(* Logix 5000 project; controller cal1615 1756-L62 rev 20.19; software revision 20.05; part 58 of 82 *)
(* tags used below, declared in another part *)
   FAULT : BOOL;   // Fault AFI
   p01_recipe_active : recipe;   // Active Recipe
   p01r02 : routine;   // System Misc Control
   p01r09_pb_global_reset : BOOL;   // System Modes PB: Global Fault Reset
   p24_di_edge_guide_auto : BOOL;   // Edge Control Inputs SS: Edge Guide Manual/Auto Auto
   p24_di_edge_guide_center : BOOL;   // Edge Control Inputs PB: Edge Guide Center
   p24_di_edge_guide_left : BOOL;   // Edge Control Inputs PB: Edge Guide Left
   p24_di_edge_guide_right : BOOL;   // Edge Control Inputs PB: Edge Guide Right
   p24_do_edge_guide_input_1 : BOOL;   // Edge Guide Digital Output Input 1
   p24_do_edge_guide_input_2 : BOOL;   // Edge Guide Digital Output Input 2
   p24_do_edge_guide_input_3 : BOOL;   // Edge Guide Digital Output Input 3
   p24_do_edge_guide_input_4 : BOOL;   // Edge Guide Digital Output Input 4
   p24_do_edge_guide_input_5 : BOOL;   // Edge Guide Digital Output Input 5
   p24r01 : routine;
   p24r10 : routine;   // Edge Control Edge Guide
   p24r10_edge_guide_auto_request : BOOL;   // Edge Control Edge Guide Auto Request
   p24r10_edge_guide_center_request : BOOL;   // Edge Control Edge Guide Center Request
   p24r10_edge_guide_jog_left_request : BOOL;   // Edge Control Edge Guide Jog Left Request
   p24r10_edge_guide_jog_right_request : BOOL;   // Edge Control Edge Guide Jog Right Request
   p24r10_timer_fault : TIMER[4];   // Edge Control Edge Guide Fault Delay
   p24r10_timer_warning : TIMER[4];   // Edge Control Edge Guide Warning Delay
   p25_ai_amps : DINT;   // Tension Stand 2 Analog Input TS 2 Motor Current
   p25_ai_hz : DINT;   // Tension Stand 2 Analog Input TS 2 Motor Hertz
   p25_ai_speed : REAL;   // Tension Stand 2 Inputs Sufrace Speed [fpm]
   p25_ai_torque : REAL;
   p25_ai_ts2_lc : REAL;   // System Metering Roll VFD Minimum Start Tension
   p25_di_brake : BOOL;   // Tension Stand 2 Digital Input TS2 & Slitter Brake Temperature OK
   p25_di_jog : BOOL;   // Tension Stand 2 Digital Input SS: Jog
   p25_di_jog_fwd : BOOL;   // Tension Stand 2 Digital Input PB: Jog Forward
   p25_di_jog_rev : BOOL;   // Tension Stand 2 Digital Input PB: Jog Reverse
   p25_di_run : BOOL;   // Tension Stand 2 Digital Input SS: Run
   p25_di_therm : BOOL;   // Tension Stand 2 Digital Input Motor Temperature OK
   p25_dint_to_hmi : DINT[16];   // Tension Stand 2 Dint to HMI
   p25_param_payout_speed_factor : REAL;   // Tension Stand 2 Accumulator Payout Winder Overspeed Factor 0.20 = 1.20 x Line Speed
   p25_status_word : INT;
   p25_ts2_gear_ratio : REAL;
   p25_ts2_roll_diameter_ft : REAL;
   p25r01 : routine;
   p25r02 : routine;
   p25r02_fault_exists : BOOL;
   p25r02_tension_dev_max : REAL;
   p25r02_tension_dev_min : REAL;
   p25r02_timer_fault : TIMER[4];   // Tension Stand 2 Misc Control Fault Dwell Timer
   p25r02_timer_warning : TIMER[4];   // Tension Stand 2 Misc Control Warning Dwell Timer
   p25r02_unack_fault : BOOL;   // Upper Poly Letoff Misc Control Unacknowledged Fault Exists
   p25r02_unack_warning : BOOL;   // Upper Poly Letoff Misc Control Unacknowledged Warning Exists
   p25r02_warning_exists : BOOL;
   p25r03 : routine;
   p25r03_ave_tq : REAL;
   p25r03_hz : SYS_SCP;   // Tension Stand 2 Analog Inputs SCP Hz
   p25r03_lc_input_max : REAL;
   p25r03_lc_input_min : REAL;
   p25r03_lc_output_max : REAL;
   p25r03_lc_output_min : REAL;
   p25r03_lc_scp : SYS_SCP;   // Tension Stand 2 Analog Input Load Cell Scaling
   p25r03_sample_timer : TIMER;
   p25r03_scaled_vfd_in : REAL;
   p25r03_timer_fault : TIMER[4];   // Tension Stand 2 Inputs Fault Dwell Timer
   p25r03_timer_warning : TIMER[4];   // Tension Stand 2 Inputs Warning Dwell Timer
   p25r03_tq_ave_ctrl : CONTROL;
   p25r03_tq_buffer : REAL[20];
   p25r03_tq_fifo : CONTROL;
   p25R03_ts2_vfd_rpm_to_speed : SYS_RPM_TO_SPEED;   // Tension Stand 2 Analog Input VFD RPM to Roll Surface Speed
   p25r03_unload : DINT;
   p25r03_vfd_in_scaling : SYS_SCP;
   p25r03_vfd_input_max : REAL;
   p25r03_vfd_input_min : REAL;
   p25r03_vfd_output_max : REAL;
   p25r03_vfd_output_min : REAL;
   p25r04 : routine;
   p25r05 : routine;
   p25r06 : routine;
   p25r07 : routine;
   p25r08 : routine;
   p25r09 : routine;   // Upper Poly Letoff Modes
   p25r10 : routine;
   p25r11 : routine;   // Tension Stand 2 VFD
(* P24_Edge_Control, continued *)

ROUTINE R10_Edge_Guide   (* ladder *)
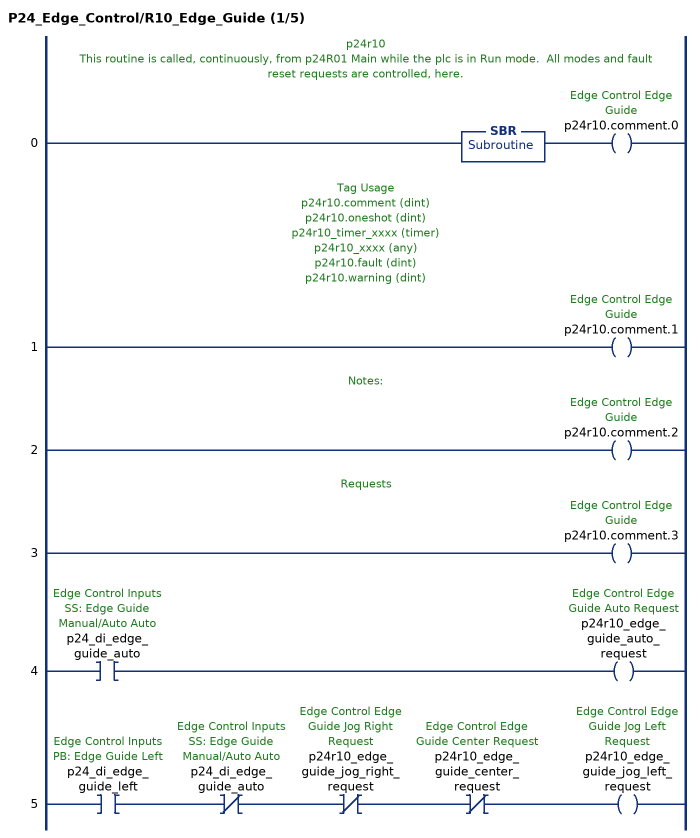
   // p24r10
   // This routine is called, continuously, from p24R01 Main while the plc is in Run mode.  All modes and fault reset requests are controlled, here.
   0: SBR()OTE(p24r10.comment.0);
   // Tag Usage
   // p24r10.comment (dint)
   // p24r10.oneshot (dint)
   // p24r10_timer_xxxx (timer)
   // p24r10_xxxx (any)
   // p24r10.fault (dint)
   // p24r10.warning (dint)
   1: OTE(p24r10.comment.1);
   // Notes:
   2: OTE(p24r10.comment.2);
   // Requests
   3: OTE(p24r10.comment.3);
   4: XIC(p24_di_edge_guide_auto)OTE(p24r10_edge_guide_auto_request);
   5: XIC(p24_di_edge_guide_left)XIO(p24_di_edge_guide_auto)XIO(p24r10_edge_guide_jog_right_request)XIO(p24r10_edge_guide_center_request)OTE(p24r10_edge_guide_jog_left_request);
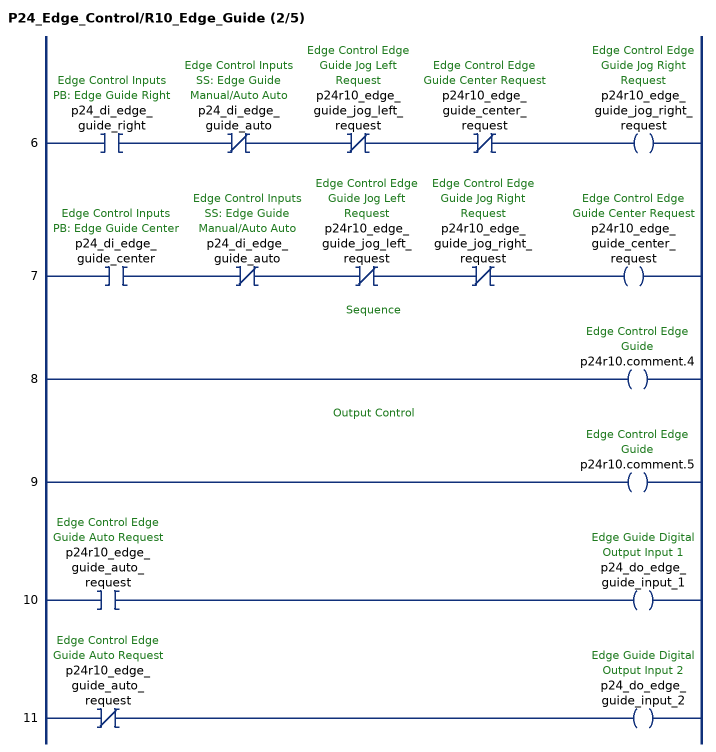
   6: XIC(p24_di_edge_guide_right)XIO(p24_di_edge_guide_auto)XIO(p24r10_edge_guide_jog_left_request)XIO(p24r10_edge_guide_center_request)OTE(p24r10_edge_guide_jog_right_request);
   7: XIC(p24_di_edge_guide_center)XIO(p24_di_edge_guide_auto)XIO(p24r10_edge_guide_jog_left_request)XIO(p24r10_edge_guide_jog_right_request)OTE(p24r10_edge_guide_center_request);
   // Sequence
   8: OTE(p24r10.comment.4);
   // Output Control
   9: OTE(p24r10.comment.5);
   10: XIC(p24r10_edge_guide_auto_request)OTE(p24_do_edge_guide_input_1);
   11: XIO(p24r10_edge_guide_auto_request)OTE(p24_do_edge_guide_input_2);
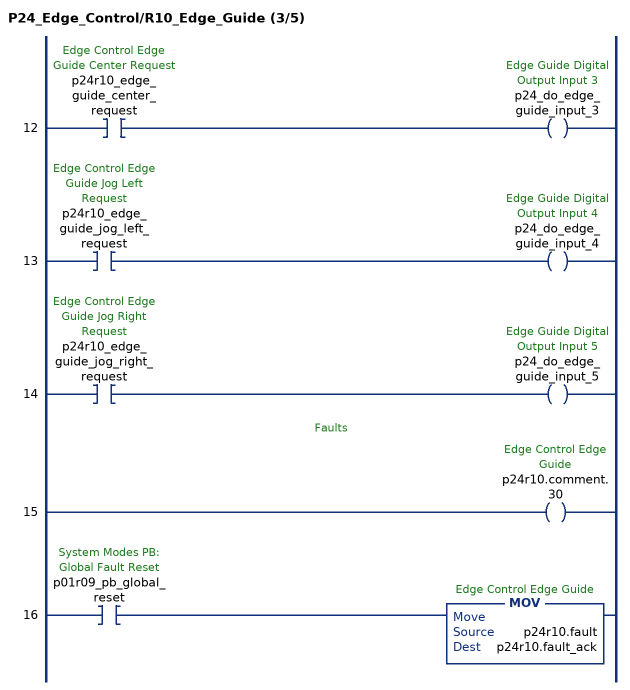
   12: XIC(p24r10_edge_guide_center_request)OTE(p24_do_edge_guide_input_3);
   13: XIC(p24r10_edge_guide_jog_left_request)OTE(p24_do_edge_guide_input_4);
   14: XIC(p24r10_edge_guide_jog_right_request)OTE(p24_do_edge_guide_input_5);
   // Faults
   15: OTE(p24r10.comment.30);
   16: XIC(p01r09_pb_global_reset)MOV(p24r10.fault,p24r10.fault_ack);
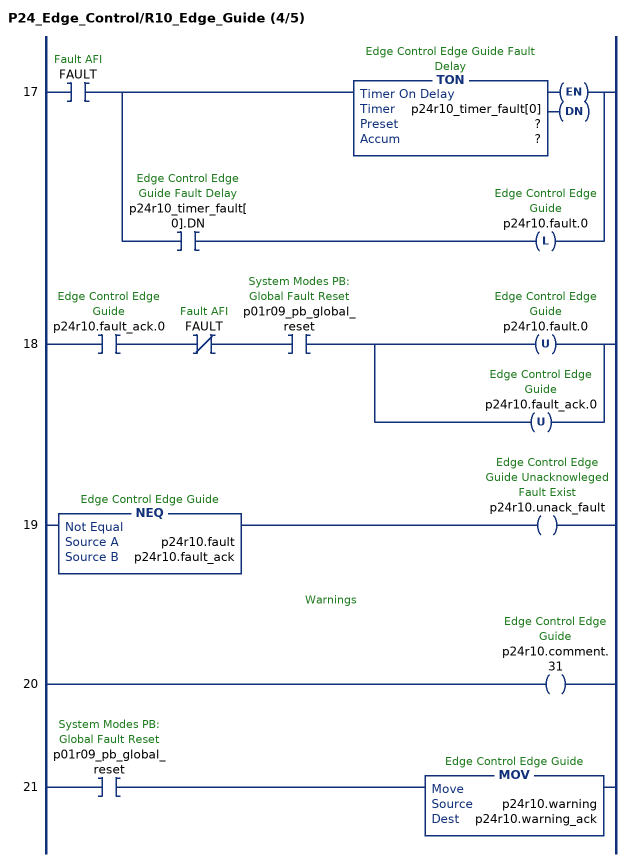
   17: XIC(FAULT)[TON(p24r10_timer_fault[0],?,?) ,XIC(p24r10_timer_fault[0].DN) OTL(p24r10.fault.0) ];
   18: XIC(p24r10.fault_ack.0)XIO(FAULT)XIC(p01r09_pb_global_reset)[OTU(p24r10.fault.0) ,OTU(p24r10.fault_ack.0) ];
   19: NEQ(p24r10.fault,p24r10.fault_ack)OTE(p24r10.unack_fault);
   // Warnings
   20: OTE(p24r10.comment.31);
   21: XIC(p01r09_pb_global_reset)MOV(p24r10.warning,p24r10.warning_ack);
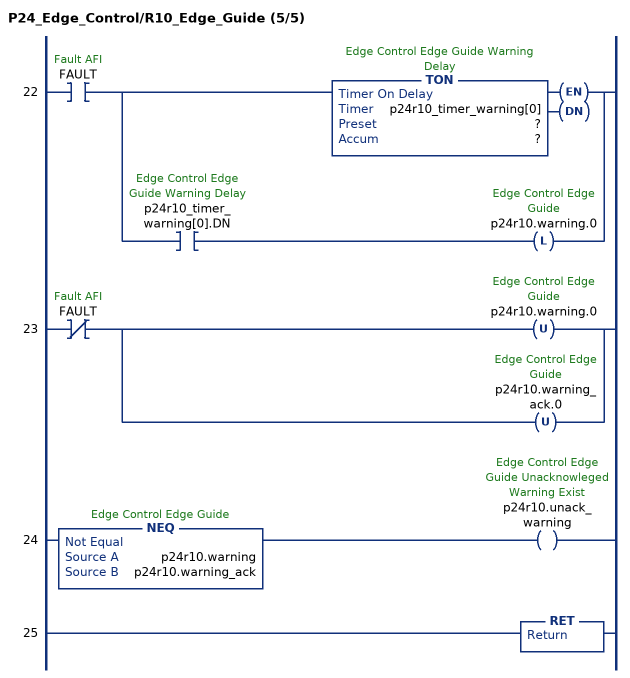
   22: XIC(FAULT)[TON(p24r10_timer_warning[0],?,?) ,XIC(p24r10_timer_warning[0].DN) OTL(p24r10.warning.0) ];
   23: XIO(FAULT)[OTU(p24r10.warning.0) ,OTU(p24r10.warning_ack.0) ];
   24: NEQ(p24r10.warning,p24r10.warning_ack)OTE(p24r10.unack_warning);
   25: RET();
END_ROUTINE
END_PROGRAM

PROGRAM P25_Tension_Stand_2   (* main routine R01_Main *)
VAR
   param_payout_speed : Setpoint := (SP := 0.2, Hi := 1.0);
   sys_limit_clamp : sys_Limit_Clamp := (max := 1.0);
END_VAR

ROUTINE R01_Main   (* ladder *)
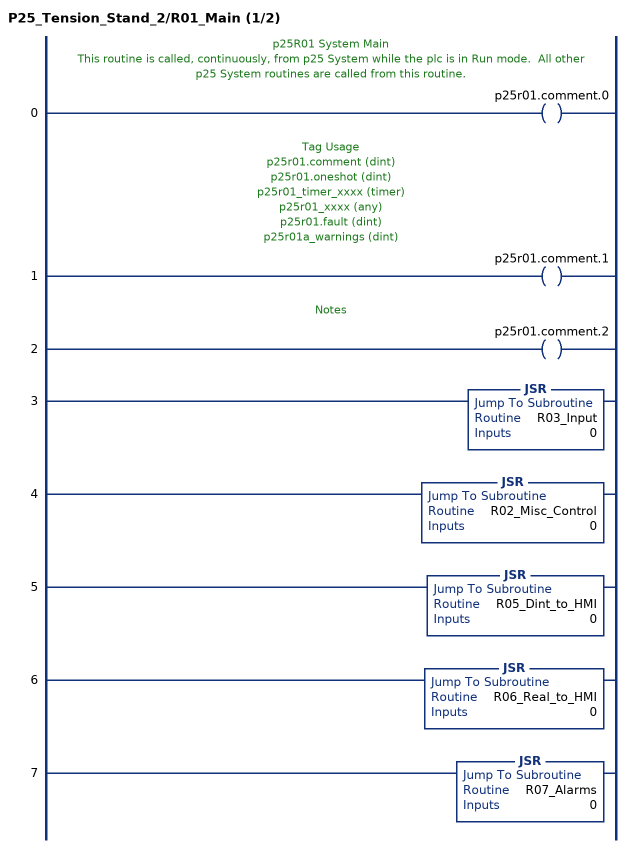
   // p25R01 System Main
   // This routine is called, continuously, from p25 System while the plc is in Run mode.  All other p25 System routines are called from this routine.
   0: OTE(p25r01.comment.0);
   // Tag Usage
   // p25r01.comment (dint)
   // p25r01.oneshot (dint)
   // p25r01_timer_xxxx (timer)
   // p25r01_xxxx (any)
   // p25r01.fault (dint)
   // p25r01a_warnings (dint)
   1: OTE(p25r01.comment.1);
   // Notes
   2: OTE(p25r01.comment.2);
   3: JSR(R03_Input,0);
   4: JSR(R02_Misc_Control,0);
   5: JSR(R05_Dint_to_HMI,0);
   6: JSR(R06_Real_to_HMI,0);
   7: JSR(R07_Alarms,0);
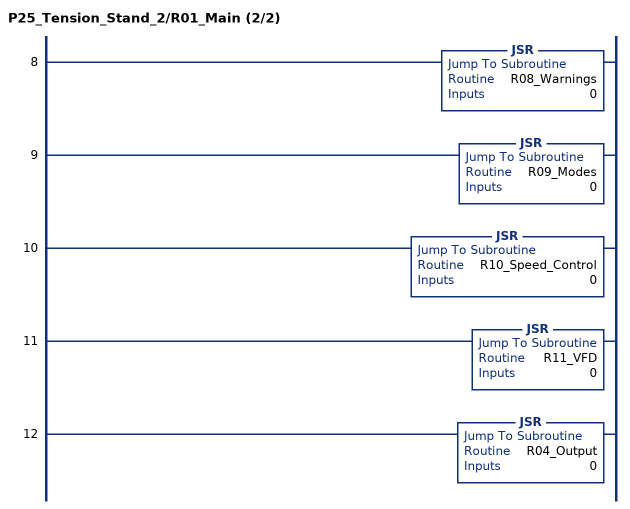
   8: JSR(R08_Warnings,0);
   9: JSR(R09_Modes,0);
   10: JSR(R10_Speed_Control,0);
   11: JSR(R11_VFD,0);
   12: JSR(R04_Output,0);
END_ROUTINE

ROUTINE R02_Misc_Control   (* ladder *)
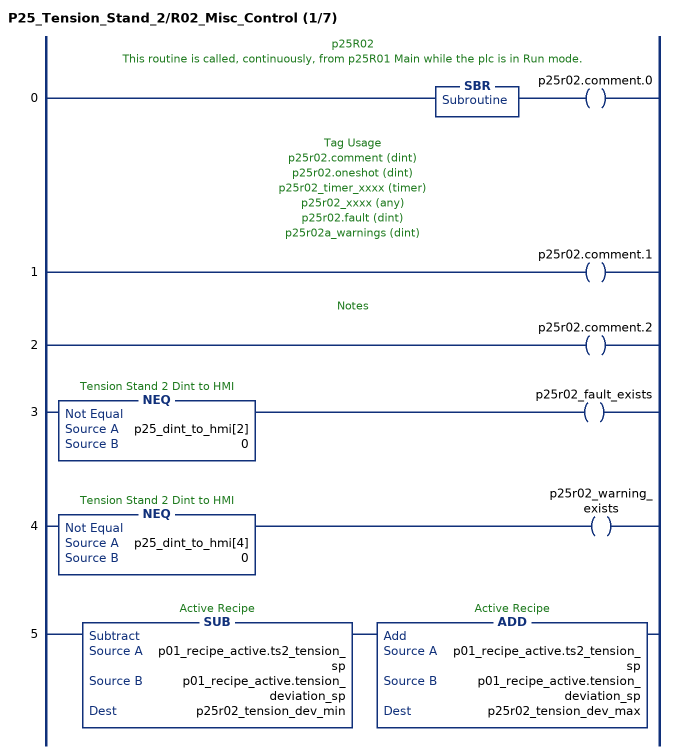
   // p25R02
   // This routine is called, continuously, from p25R01 Main while the plc is in Run mode.
   0: SBR()OTE(p25r02.comment.0);
   // Tag Usage
   // p25r02.comment (dint)
   // p25r02.oneshot (dint)
   // p25r02_timer_xxxx (timer)
   // p25r02_xxxx (any)
   // p25r02.fault (dint)
   // p25r02a_warnings (dint)
   1: OTE(p25r02.comment.1);
   // Notes
   2: OTE(p25r02.comment.2);
   3: NEQ(p25_dint_to_hmi[2],0)OTE(p25r02_fault_exists);
   4: NEQ(p25_dint_to_hmi[4],0)OTE(p25r02_warning_exists);
   5: SUB(p01_recipe_active.ts2_tension_sp,p01_recipe_active.tension_deviation_sp,p25r02_tension_dev_min)ADD(p01_recipe_active.ts2_tension_sp,p01_recipe_active.tension_deviation_sp,p25r02_tension_dev_max);
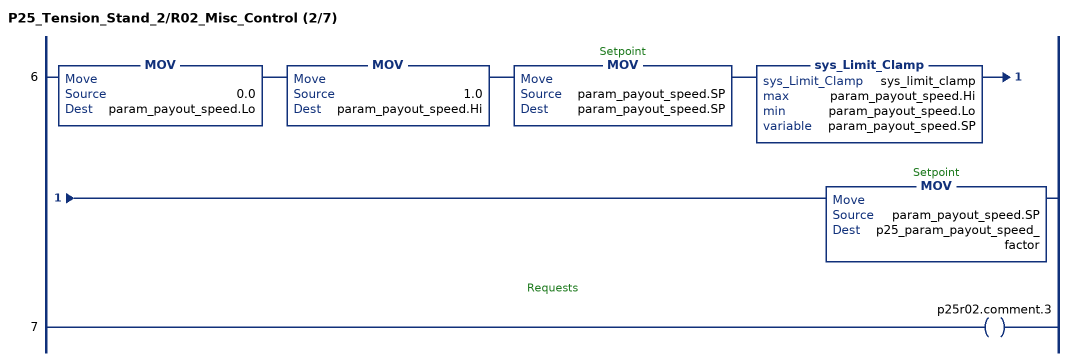
   6: MOV(0.0,param_payout_speed.Lo)MOV(1.0,param_payout_speed.Hi)MOV(param_payout_speed.SP,param_payout_speed.SP)sys_Limit_Clamp(sys_limit_clamp,param_payout_speed.Hi,param_payout_speed.Lo,param_payout_speed.SP)MOV(param_payout_speed.SP,p25_param_payout_speed_factor);
   // Requests
   7: OTE(p25r02.comment.3);
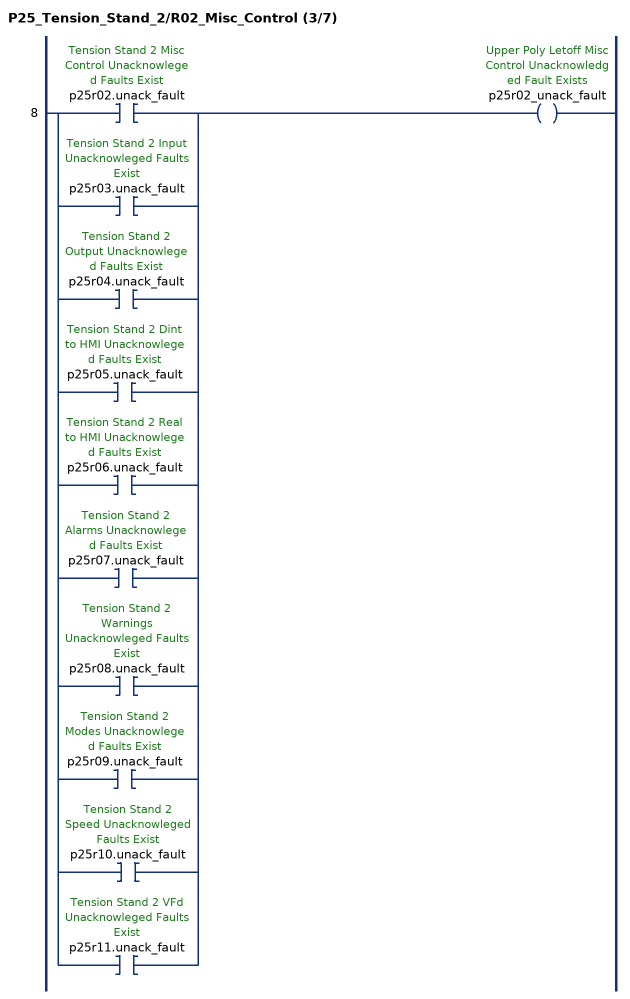
   8: [XIC(p25r02.unack_fault) ,XIC(p25r03.unack_fault) ,XIC(p25r04.unack_fault) ,XIC(p25r05.unack_fault) ,XIC(p25r06.unack_fault) ,XIC(p25r07.unack_fault) ,XIC(p25r08.unack_fault) ,XIC(p25r09.unack_fault) ,XIC(p25r10.unack_fault) ,XIC(p25r11.unack_fault) ]OTE(p25r02_unack_fault);
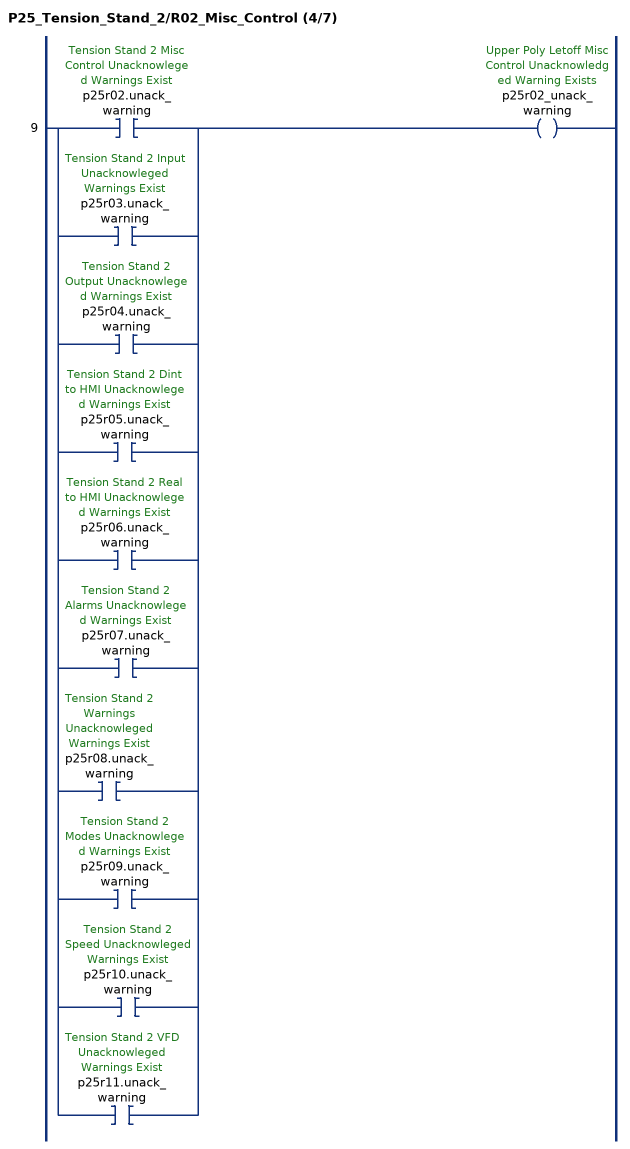
   9: [XIC(p25r02.unack_warning) ,XIC(p25r03.unack_warning) ,XIC(p25r04.unack_warning) ,XIC(p25r05.unack_warning) ,XIC(p25r06.unack_warning) ,XIC(p25r07.unack_warning) ,XIC(p25r08.unack_warning) ,XIC(p25r09.unack_warning) ,XIC(p25r10.unack_warning) ,XIC(p25r11.unack_warning) ]OTE(p25r02_unack_warning);
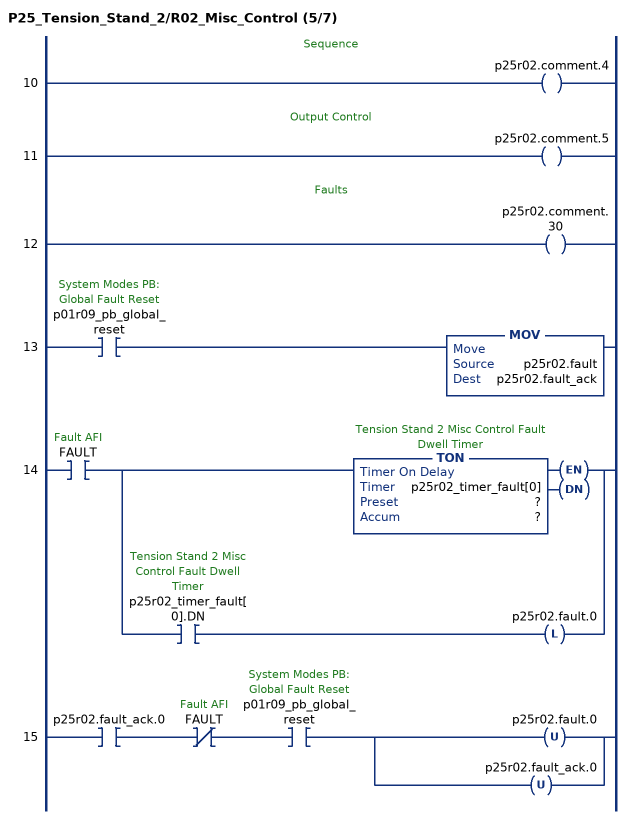
   // Sequence
   10: OTE(p25r02.comment.4);
   // Output Control
   11: OTE(p25r02.comment.5);
   // Faults
   12: OTE(p25r02.comment.30);
   13: XIC(p01r09_pb_global_reset)MOV(p25r02.fault,p25r02.fault_ack);
   14: XIC(FAULT)[TON(p25r02_timer_fault[0],?,?) ,XIC(p25r02_timer_fault[0].DN) OTL(p25r02.fault.0) ];
   15: XIC(p25r02.fault_ack.0)XIO(FAULT)XIC(p01r09_pb_global_reset)[OTU(p25r02.fault.0) ,OTU(p25r02.fault_ack.0) ];
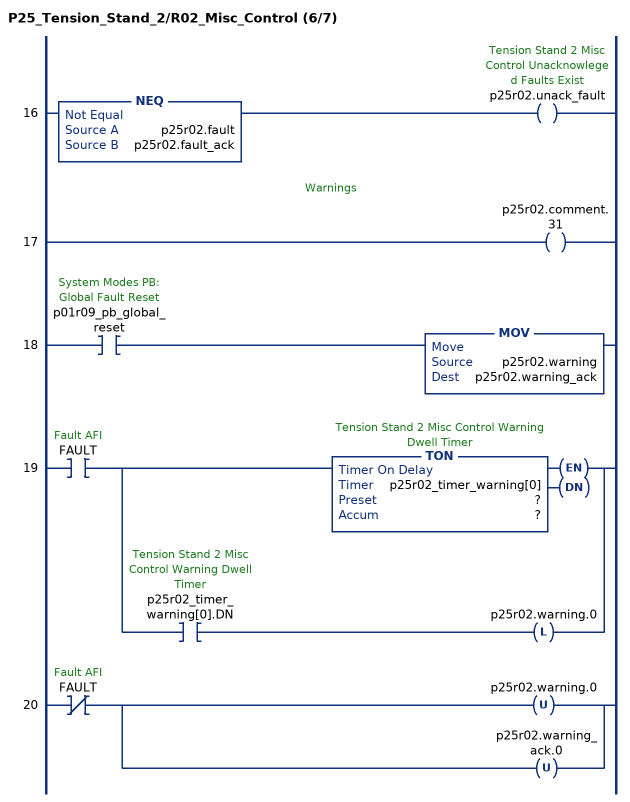
   16: NEQ(p25r02.fault,p25r02.fault_ack)OTE(p25r02.unack_fault);
   // Warnings
   17: OTE(p25r02.comment.31);
   18: XIC(p01r09_pb_global_reset)MOV(p25r02.warning,p25r02.warning_ack);
   19: XIC(FAULT)[TON(p25r02_timer_warning[0],?,?) ,XIC(p25r02_timer_warning[0].DN) OTL(p25r02.warning.0) ];
   20: XIO(FAULT)[OTU(p25r02.warning.0) ,OTU(p25r02.warning_ack.0) ];
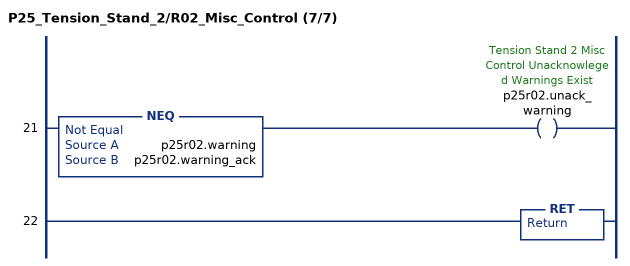
   21: NEQ(p25r02.warning,p25r02.warning_ack)OTE(p25r02.unack_warning);
   22: RET();
END_ROUTINE

ROUTINE R03_Input   (* ladder *)
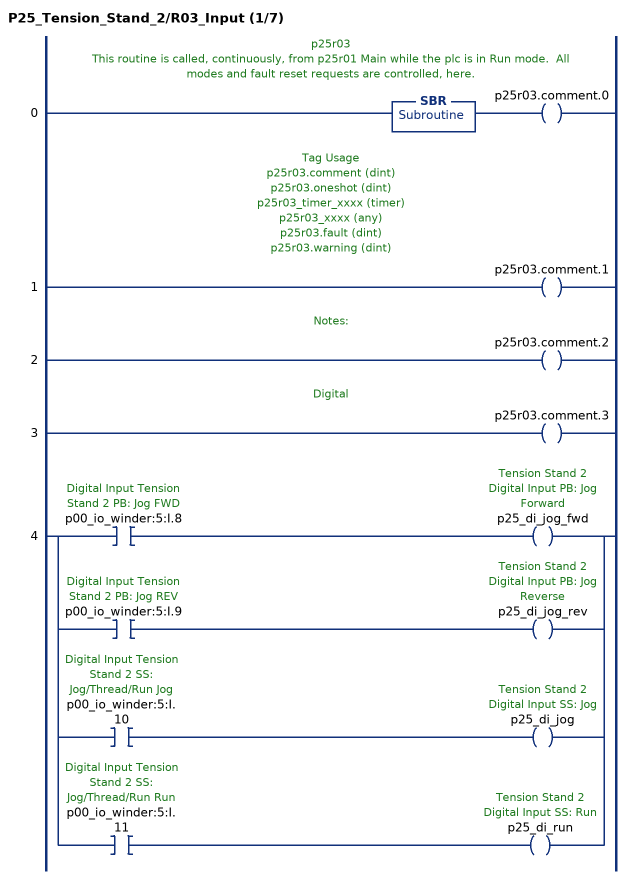
   // p25r03
   // This routine is called, continuously, from p25r01 Main while the plc is in Run mode.  All modes and fault reset requests are controlled, here.
   0: SBR()OTE(p25r03.comment.0);
   // Tag Usage
   // p25r03.comment (dint)
   // p25r03.oneshot (dint)
   // p25r03_timer_xxxx (timer)
   // p25r03_xxxx (any)
   // p25r03.fault (dint)
   // p25r03.warning (dint)
   1: OTE(p25r03.comment.1);
   // Notes:
   2: OTE(p25r03.comment.2);
   // Digital
   3: OTE(p25r03.comment.3);
   4: [XIC(p00_io_winder:5:I.8) OTE(p25_di_jog_fwd) ,XIC(p00_io_winder:5:I.9) OTE(p25_di_jog_rev) ,XIC(p00_io_winder:5:I.10) OTE(p25_di_jog) ,XIC(p00_io_winder:5:I.11) OTE(p25_di_run) ];
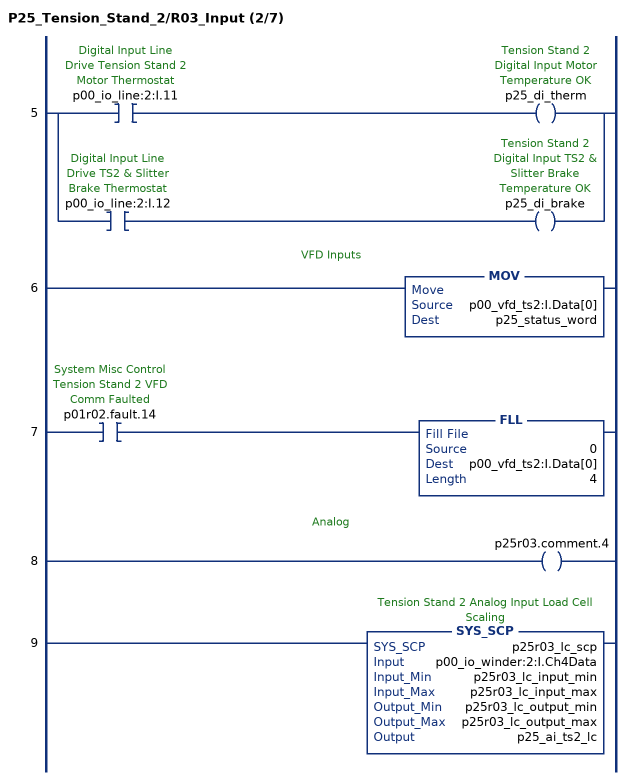
   5: [XIC(p00_io_line:2:I.11) OTE(p25_di_therm) ,XIC(p00_io_line:2:I.12) OTE(p25_di_brake) ];
   // VFD Inputs
   6: MOV(p00_vfd_ts2:I.Data[0],p25_status_word);
   7: XIC(p01r02.fault.14)FLL(0,p00_vfd_ts2:I.Data[0],4);
   // Analog
   8: OTE(p25r03.comment.4);
   9: SYS_SCP(p25r03_lc_scp,p00_io_winder:2:I.Ch4Data,p25r03_lc_input_min,p25r03_lc_input_max,p25r03_lc_output_min,p25r03_lc_output_max,p25_ai_ts2_lc);
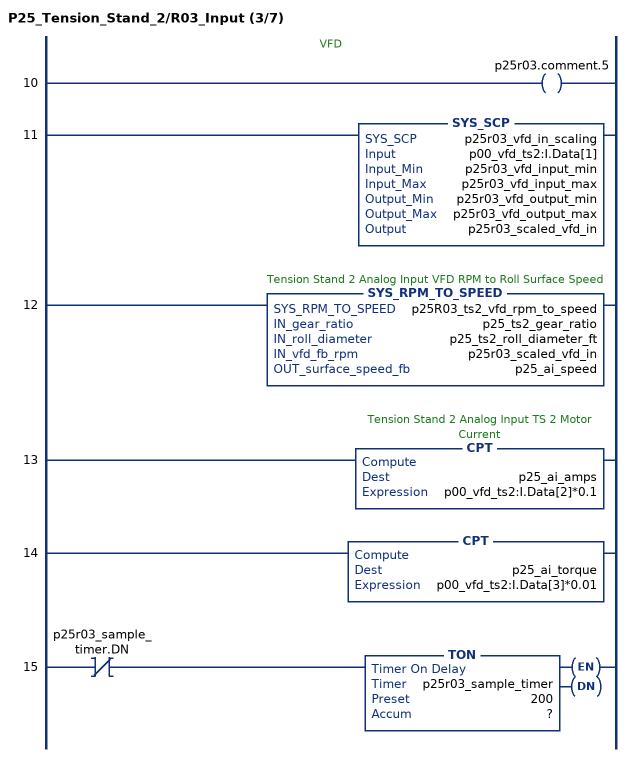
   // VFD
   10: OTE(p25r03.comment.5);
   11: SYS_SCP(p25r03_vfd_in_scaling,p00_vfd_ts2:I.Data[1],p25r03_vfd_input_min,p25r03_vfd_input_max,p25r03_vfd_output_min,p25r03_vfd_output_max,p25r03_scaled_vfd_in);
   12: SYS_RPM_TO_SPEED(p25R03_ts2_vfd_rpm_to_speed,p25_ts2_gear_ratio,p25_ts2_roll_diameter_ft,p25r03_scaled_vfd_in,p25_ai_speed);
   13: CPT(p25_ai_amps,p00_vfd_ts2:I.Data[2]*0.1);
   14: CPT(p25_ai_torque,p00_vfd_ts2:I.Data[3]*0.01);
   15: XIO(p25r03_sample_timer.DN)TON(p25r03_sample_timer,?,?);
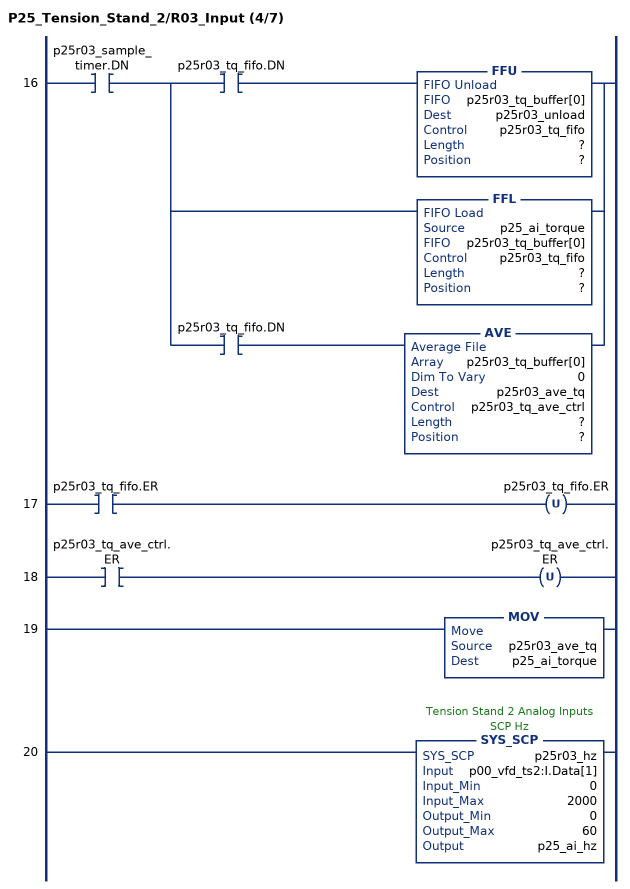
   16: XIC(p25r03_sample_timer.DN)[XIC(p25r03_tq_fifo.DN) FFU(p25r03_tq_buffer[0],p25r03_unload,p25r03_tq_fifo,?,?) ,FFL(p25_ai_torque,p25r03_tq_buffer[0],p25r03_tq_fifo,?,?) ,XIC(p25r03_tq_fifo.DN) AVE(p25r03_tq_buffer[0],0,p25r03_ave_tq,p25r03_tq_ave_ctrl,?,?) ];
   17: XIC(p25r03_tq_fifo.ER)OTU(p25r03_tq_fifo.ER);
   18: XIC(p25r03_tq_ave_ctrl.ER)OTU(p25r03_tq_ave_ctrl.ER);
   19: MOV(p25r03_ave_tq,p25_ai_torque);
   20: SYS_SCP(p25r03_hz,p00_vfd_ts2:I.Data[1],0,2000,0,60,p25_ai_hz);
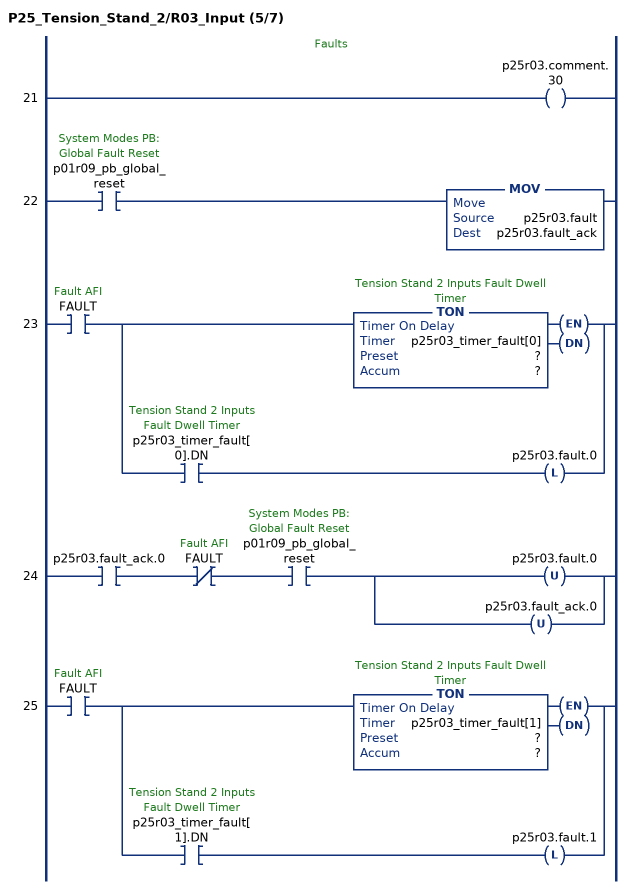
   // Faults
   21: OTE(p25r03.comment.30);
   22: XIC(p01r09_pb_global_reset)MOV(p25r03.fault,p25r03.fault_ack);
   23: XIC(FAULT)[TON(p25r03_timer_fault[0],?,?) ,XIC(p25r03_timer_fault[0].DN) OTL(p25r03.fault.0) ];
   24: XIC(p25r03.fault_ack.0)XIO(FAULT)XIC(p01r09_pb_global_reset)[OTU(p25r03.fault.0) ,OTU(p25r03.fault_ack.0) ];
   25: XIC(FAULT)[TON(p25r03_timer_fault[1],?,?) ,XIC(p25r03_timer_fault[1].DN) OTL(p25r03.fault.1) ];
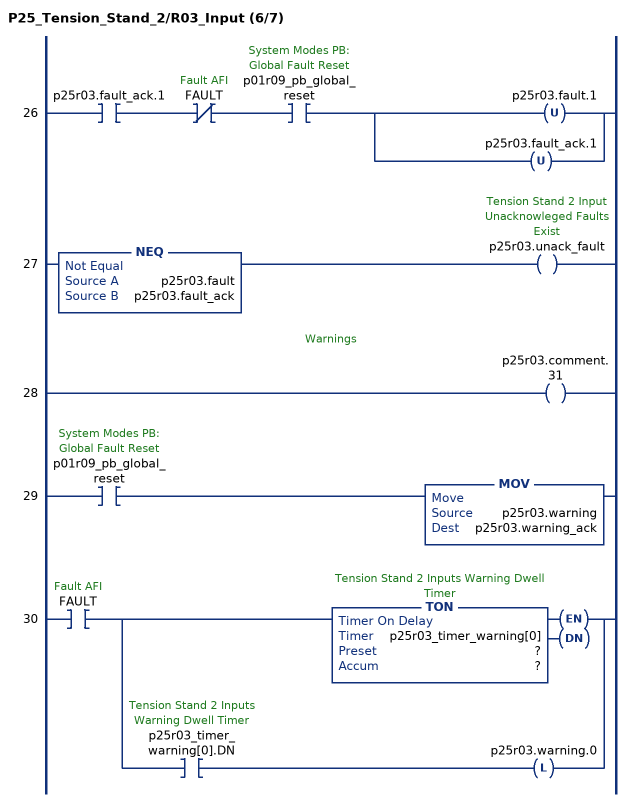
   26: XIC(p25r03.fault_ack.1)XIO(FAULT)XIC(p01r09_pb_global_reset)[OTU(p25r03.fault.1) ,OTU(p25r03.fault_ack.1) ];
   27: NEQ(p25r03.fault,p25r03.fault_ack)OTE(p25r03.unack_fault);
   // Warnings
   28: OTE(p25r03.comment.31);
   29: XIC(p01r09_pb_global_reset)MOV(p25r03.warning,p25r03.warning_ack);
   30: XIC(FAULT)[TON(p25r03_timer_warning[0],?,?) ,XIC(p25r03_timer_warning[0].DN) OTL(p25r03.warning.0) ];
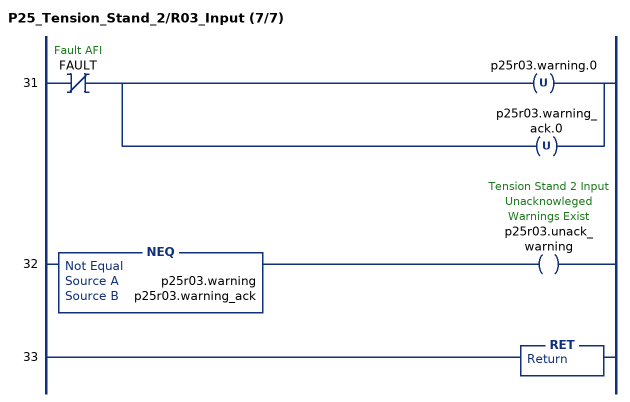
   31: XIO(FAULT)[OTU(p25r03.warning.0) ,OTU(p25r03.warning_ack.0) ];
   32: NEQ(p25r03.warning,p25r03.warning_ack)OTE(p25r03.unack_warning);
   33: RET();
END_ROUTINE
